// TIA Portal V16 export
// export: Created 2021-11-12T13:32:24.5573668Z, ExportSetting WithDefaults, DisplayName Totally Integrated Automation Portal, DisplayVersion V16 Update 3, DisplayName TIA Portal Version Control Interface, DisplayVersion V16 Update 2, DisplayName TIA Portal Openness, DisplayVersion V16 Update 3, DisplayName SINAMICS Startdrive Advanced, DisplayVersion V16 Update 5, DisplayName SINAMICS Startdrive G130, G150, S120, S150, SINAMICS MV, S210, DisplayVersion V16 Update 5, DisplayName SINAMICS Startdrive G110M, G120, G120C, G120D, G120P, G115D, DisplayVersion V16 Update 5, DisplayName STEP 7 Professional, DisplayVersion V16 Update 3, DisplayName STEP 7 Safety, DisplayVersion V16, DisplayName WinCC UA Professional, DisplayVersion V16 Update 3
DATA_BLOCK "IDB_StationKAS2"   // DB169
{ DB_Accessible_From_OPC_UA := 'FALSE' }
VERSION : 0.1
// stored: AutoNumber true, DBAccessibleFromOPCUA false, InstanceOfName StationKAS2, InstanceOfType FB
"StationKAS2"
   // VAR_INPUT
   //    IS_Inputs : "UDT_COMM_KAS2_CRS";
   // END_VAR
   // VAR_OUTPUT
   //    OS_Outputs : "UDT_COMM_CRS_KAS2";
   // END_VAR
   // VAR
   //    SF_Alarm1 : "STD_DI_Mon";
   //    SF_Alarm2 { S7_SetPoint := 'True'} : "STD_DI_Mon";
   //    SF_PartOk { S7_SetPoint := 'True'} : "STD_PartCounter";
   //    SF_PartNok { S7_SetPoint := 'True'} : "STD_PartCounter";
   //    SS_Edge : Array[0..15] of Bool;
   // END_VAR
BEGIN
END_DATA_BLOCK
